# EPICS autosave request: pylonApp/Db/pylon_settings.req
file "ADGenICam_settings.req", P=$(P), R=$(R)
$(P)$(R)TimeStampMode
$(P)$(R)UniqueIdMode
$(P)$(R)ConvertPixelFormat
$(P)$(R)ConvertBitAlign
$(P)$(R)ConvertShiftBits
